{attribute 'OPC.UA.DA.StructuredType' := '1'}
FUNCTION_BLOCK FB_Sensor_GrowMedium_PH EXTENDS FB_BaseSensor IMPLEMENTS I_Device, I_Sensor

VAR

	bCAL: BOOL := FALSE;
	eSMState: (WAIT, CAL_4, CAL_7, CALC_CORRECTION) := WAIT;
	
END_VAR
	
VAR PERSISTENT 

	nPH4_val: REAL;
	nPH7_val: REAL;
	
	b4High_0_20High_1: BOOL := TRUE;
	
	nCurveGradient: REAL := 6.0/16.0; // Sensor range is PH 3 to 9 over 16mA range (4-20mA)
	nCurveOffset: REAL := 1.5; 
END_VAR

calculate();
filter();

// Detect if any buttons in ignition have been pressed for Calibration
IF bCAL THEN 
	bCAL := FALSE;
	CASE eSMState OF
		WAIT:
			eSMState := CAL_4;
		CAL_4:
			eSMState := CAL_7;
		CAL_7:
			eSMState := CALC_CORRECTION;
	END_CASE
END_IF




CASE eSMState OF 
	WAIT:
		// wait here for a calibration command to be received
		eState := E_DeviceState.RUNNING;
		
	CAL_4:
		nPH4_val := nFilteredCurrent;
		eState := E_DeviceState.CAL_STEP1;

	CAL_7:
		nPH7_val := nFilteredCurrent;
		eState := E_DeviceState.CAL_STEP2;

	CALC_CORRECTION:
		nCurveGradient := 3.0 / (nPH7_val - nPH4_val);
		nCurveOffset := 4.0 - (nCurveGradient * nPH4_val);
		eState := E_DeviceState.CAL_STEP3;
		eSMState := WAIT;
		
END_CASE

METHOD PRIVATE calculate : BOOL
VAR_INPUT
	
END_VAR
IF b4High_0_20High_1 THEN
	nMeasuredCurrent := (INT_TO_REAL(nRawInput)/GVL.nMaxADCOutput)*16.0 + 4.0; // in mA
ELSE
	nMeasuredCurrent := 20.0 - (INT_TO_REAL(nRawInput)/GVL.nMaxADCOutput)*16.00; 
END_IF


// nCurrentValue := (nCurveGradient * nMeasuredCurrent) + nCurveOffset; 

nCurrentValue := (nCurveGradient * nFilteredCurrent) + nCurveOffset; // delete this eventually

nCurrentValueFiltered := (nCurveGradient * nFilteredCurrent) + nCurveOffset;
END_METHOD

METHOD calibrate : BOOL
VAR_INPUT
	
END_VAR

bCAL := TRUE;
END_METHOD

{warning 'add method implementation '}
METHOD disable : BOOL
bEnable := FALSE;
END_METHOD

{warning 'add method implementation '}
METHOD enable : BOOL
bEnable := TRUE;
END_METHOD

{warning 'add method implementation '}
METHOD FB_init : BOOL
VAR_INPUT
	(* if TRUE, the retain variables are initialized (warm start / cold start)*)
	bInitRetains	: BOOL;
	(* if TRUE, the instance afterwards gets moved into the copy code (online change)*)
	bInCopyCode	: BOOL;
	
	SensorID	: STRING(80);
	SensorDescr	: STRING(255);
	SensorType	: E_SensorType;
END_VAR
sID := SensorID;
sDescr := SensorDescr;
eSensorType := SensorType;
END_METHOD

{warning 'add method implementation '}
METHOD getType : E_SensorType
getType := eSensorType;
END_METHOD

{warning 'add method implementation '}
METHOD getValue : REAL
getValue := nCurrentValue;
END_METHOD

{warning 'add method implementation '}
METHOD write : BOOL
// use this method to initiated a hardware read from assigned IO if required
END_METHOD

END_FUNCTION_BLOCK

(* stored: Version 1.1.0.1, ProductVersion 3.1.4024.12
   POU FB_Sensor_GrowMedium_PH: Id {2e6af340-be58-481e-a17f-47bf14761533}, SpecialFunc None
   Method calculate: Id {1a21ea4a-7185-40e5-ad12-271de796c1a1}
   Method calibrate: Id {dd904280-ebf4-4cf1-b716-1fbeb3afc91c}
   Method disable: Id {6f830881-a44e-482d-82ba-5b0a54100606}
   Method enable: Id {ea4edaef-daa0-42ea-b0fb-0ddd0b2409a5}
   Method FB_init: Id {0fadeb0e-12ef-405e-836e-045e66683241}
   Method getType: Id {bef06be2-6fd2-4d79-af65-7e7716e0d616}
   Method getValue: Id {0738a069-70e3-49a3-bcf0-ce82822f4b5e}
   Method write: Id {c8bf41da-8610-4c78-805f-b1668d4312ec} *)
